KUKA KRL data list: Station2.dat

&ACCESS RVE
DEFDAT  Station2 PUBLIC

ENDDAT
